PROGRAM MAIN
VAR
	bStartPB  : BOOL;
	bEndPB :	BOOL	;
END_VAR

END_PROGRAM

(* stored: Version 1.1.0.1, ProductVersion 3.1.4024.12
   POU MAIN: Id {f7277d4d-042a-419c-aaaa-0a9b34d5f3cc}, SpecialFunc None *)
